FUNCTION_BLOCK StateBuffer
VAR_GENERIC CONSTANT
	nMax				: UDINT(0..16#FFFFFFE) := 1;
END_VAR
IMPLEMENTS I_StateBuffer
VAR
	_iState				: ARRAY[0..nMax] OF I_State;
	_nHead				: UDINT;
	_nTail				: UDINT;
	_nLen				: UDINT;

	
	_fbTagOwner			: Tags.TagOwner;
END_VAR

METHOD Cap : UDINT
VAR_INPUT
END_VAR
Cap := nMax;
END_METHOD

METHOD Length : UDINT
VAR_INPUT
END_VAR
Length := _nLen;
END_METHOD

METHOD Pop : Results.Result
VAR_OUTPUT
	iState			: I_State;
END_VAR
IF _nHead = _nTail THEN
    Pop := Results.None;
    RETURN;
END_IF

iState := _iState[_nHead];
_iState[_nHead] := 0;

_nHead := _nHead + 1;
_nLen := _nLen - 1;

IF _nHead > nMax THEN
    _nHead := 0;
END_IF

Pop := Results.Ok;
END_METHOD

METHOD Push : Results.Result
VAR_INPUT
	iState			: I_State;
END_VAR
VAR
	_nNextTail 		: UDINT;
END_VAR
IF iState = 0 THEN
	Push := Results.Err.Itf0;
	RETURN;
END_IF

_nNextTail := _nTail + 1;

IF _nNextTail > nMax THEN
    _nNextTail := 0;
END_IF

IF _nNextTail = _nHead THEN
    Push := Results.Err.Ovf; 
    RETURN;
END_IF

_nLen := _nLen + 1;
_iState[_nTail] := iState;
_nTail := _nNextTail;
Push := Results.Ok;
END_METHOD

END_FUNCTION_BLOCK

(* stored: Version 1.1.0.1
   POU StateBuffer: Id {c72b10a5-ebed-4e92-a090-567cf79b812e}, SpecialFunc None
   Folder Other: Id {9e7ac76f-4d0e-4ca5-8870-fa5600f9c22c}
   Folder Push: Id {fca17cab-fb89-4124-bdc0-545fbd4443f5}
   Method Cap: Id {cd19f415-bdc0-4a48-be4d-06e0fa03966e}
   Method Length: Id {8357a420-23aa-4183-9087-bb8cd5148145}
   Method Pop: Id {722c1396-ea3f-4454-a3a0-4804c31d5645}
   Method Push: Id {9d46582f-4419-4027-8c47-8930019ed874} *)
